// TIA Portal V20 export
DATA_BLOCK "DB_Alarm"   // DB16
// stored: Access Published, MemoryReserve 100, Namespace PackedLine
   VAR
      "word" : Struct
         Line : Struct
            PackedLine : Struct
               Conveyor : Array[_.minPackedLine.._.maxPackedLine] of Word;
            END_STRUCT;
         END_STRUCT;
      END_STRUCT;
   END_VAR
BEGIN
END_DATA_BLOCK
